// TIA Portal V18 export
FUNCTION "selection_Machine" : Void   // FC1, LAD
{ S7_Optimized_Access := 'TRUE' }
VERSION : 0.1
// stored: AutoNumber true, IsIECCheckEnabled false, SetENOAutomatically false, UDAEnableTagReadback false
BEGIN

REGION Network 1 (SCL)
   IF "selection_machie_db"."1k_2k" = TRUE THEN
       "Mixing ratio"."Mixing ratio set" := 0;
   END_IF;
END_REGION
END_FUNCTION
